{attribute 'strict'}
//Pathing Enum
TYPE E_OutletNumber :
(
	Outlet_2:=1,
    Outlet_1:= 2,
    Recirculation:=3
)USINT;
END_TYPE

(* stored: Version 1.1.0.1
   DUT E_OutletNumber: Id {56cd93e0-eb0f-42d8-85b9-e404dce89284} *)
